PROGRAM Pine_Branch_Test
VAR
END_VAR

// Pine branch test by Alan from his laptop.

END_PROGRAM

(* stored: Version 1.1.0.1, ProductVersion 3.1.4024.11
   POU Pine_Branch_Test: Id {bdfe5762-88cd-45bf-898f-fd5def4aba6d}, SpecialFunc None *)
